// Mitsubishi GX Works2 project: k01   PLC: Q02/Q02H

PROGRAM MAIN
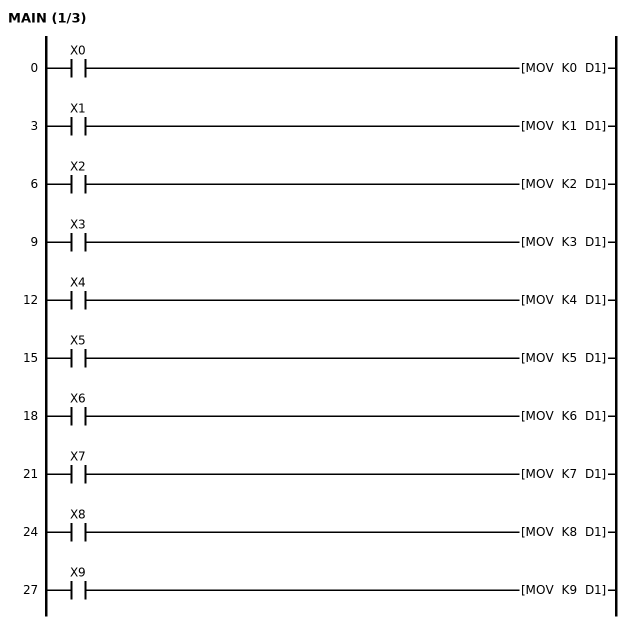
0     LD      X0
      MOV     K0 D1
3     LD      X1
      MOV     K1 D1
6     LD      X2
      MOV     K2 D1
9     LD      X3
      MOV     K3 D1
12    LD      X4
      MOV     K4 D1
15    LD      X5
      MOV     K5 D1
18    LD      X6
      MOV     K6 D1
21    LD      X7
      MOV     K7 D1
24    LD      X8
      MOV     K8 D1
27    LD      X9
      MOV     K9 D1
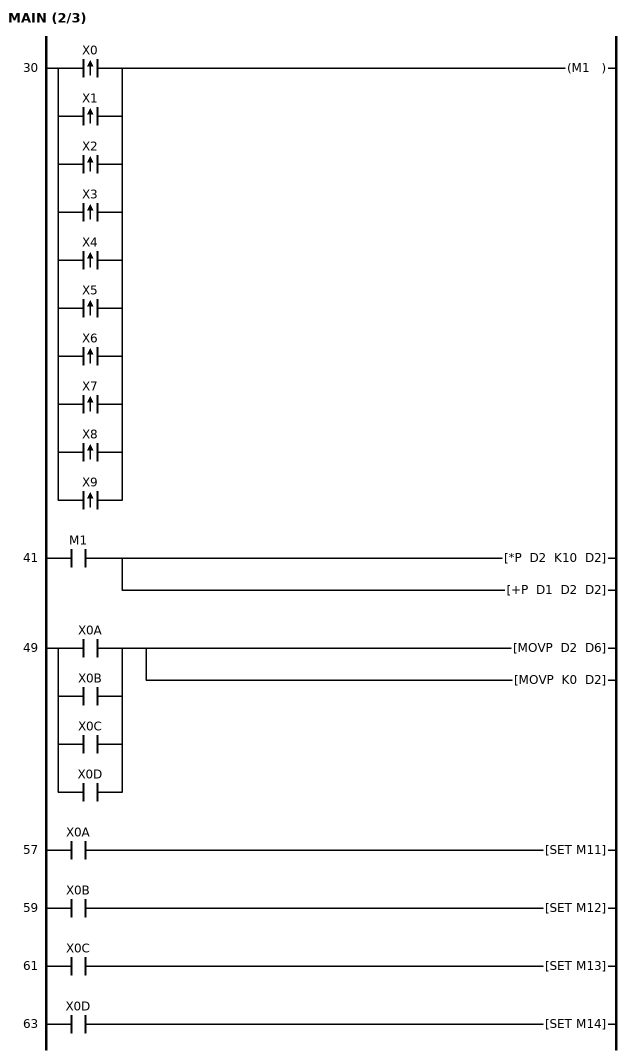
30    LDP     X0
      ORP     X1
      ORP     X2
      ORP     X3
      ORP     X4
      ORP     X5
      ORP     X6
      ORP     X7
      ORP     X8
      ORP     X9
      OUT     M1
41    LD      M1
      *P      D2 K10 D2
      +P      D1 D2 D2
49    LD      X0A
      OR      X0B
      OR      X0C
      OR      X0D
      MOVP    D2 D6
      MOVP    K0 D2
57    LD      X0A
      SET     M11
59    LD      X0B
      SET     M12
61    LD      X0C
      SET     M13
63    LD      X0D
      SET     M14
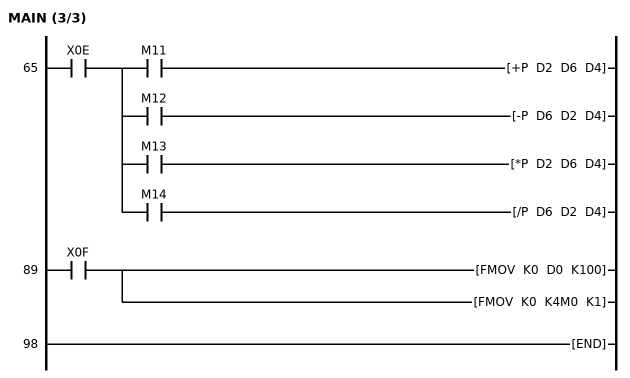
65    LD      X0E
      MPS
      AND     M11
      +P      D2 D6 D4
      MRD
      AND     M12
      -P      D6 D2 D4
      MRD
      AND     M13
      *P      D2 D6 D4
      MPP
      AND     M14
      /P      D6 D2 D4
89    LD      X0F
      FMOV    K0 D0 K100
      FMOV    K0 K4M0 K1
98    END
END_PROGRAM
